{attribute 'GeneratedUsingTerminal: EK1122-0000-0018'}
{attribute addProperty BoxType "EK1122-0000-0018"}
{attribute addProperty Id "Beckhoff_EM3xxxsub_EK1100EK1100_AB5A94672"}
{attribute addProperty CRC "281876091"}
{attribute addProperty Size "2"}
TYPE Beckhoff_EM3xxxEK1122_10CD167B EXTENDS EK1122_AB5A9467 :
STRUCT
	{attribute addProperty Name "Beckhoff_EM3xxxsub_EK1100"}
	{attribute addProperty PreviousPort "Beckhoff EM3xxxEK1122 : D"}
	Beckhoff_EM3xxxsub_EK1100 : EK1100_AB5A9467;
END_STRUCT
END_TYPE

(* stored: Version 1.2.0.0, ProductVersion 3.1.4024.9
   DUT Beckhoff_EM3xxxEK1122_10CD167B: Id {2fc235b0-0efd-4dfc-b5e3-9675b6931813} *)
